(* IEC 61131-3 sources: SJ_AGV/PLC/Standard_functions.4.4.0/Navigation, 2 files *)

(* ---- LS2000_FB.ST ---- *)
FUNCTION_BLOCK LS2000_FB
VAR_EXTERNAL
	NDC8 : NDC8_T;
END_VAR

VAR_INPUT

END_VAR

VAR_OUTPUT
	Slowdown : bool;
END_VAR

VAR
	LS2000Field1TON :TON;
	LS2000Field2TON :TON;
END_VAR
(* Function to slow down, and eventually stop, if there is an obstacle in the path of the LS2000. *)

LS2000Field1TON (IN:= NDC8.LS2000.Field1_Triggered, PT:=T#160ms); (*Timer 160ms to filter signal*)
LS2000Field2TON (IN:= NDC8.LS2000.Field2_Triggered, PT:=T#160ms); (*Timer 160ms to filter signal *)

(* Stop window (Field 1), relative the scanner. *)
NDC8.LS2000.Field1_X1 := NDC8.LS2000.X - 100;	(* 500 mm behind. 		*)
NDC8.LS2000.Field1_X2 := NDC8.LS2000.X + 100;	(* 500 mm in front. 	*)
NDC8.LS2000.Field1_Y1 := NDC8.LS2000.Y - 100;	(* 500 mm to the left. 	*)
NDC8.LS2000.Field1_Y2 := NDC8.LS2000.Y + 100;	(* 500 mm to the right. *)

(* Slow down window (Field 2), relative the scanner. *)
NDC8.LS2000.Field2_X1 := NDC8.LS2000.X - 100;	(* 1000 mm behind.		*)
NDC8.LS2000.Field2_X2 := NDC8.LS2000.X + 100;	(* 1000 mm in front.	*)
NDC8.LS2000.Field2_Y1 := NDC8.LS2000.Y - 100;	(* 1000 mm to the left.	*)
NDC8.LS2000.Field2_Y2 := NDC8.LS2000.Y + 100;	(* 1000 mm to the right.*)

if INPUT.Manual  or NDC8.LoadOperation.OperationCode <> 0 then
	NDC8.LS2000.Field1_X1 := NDC8.LS2000.X ;	(* 500 mm behind. 		*)
	NDC8.LS2000.Field1_X2 := NDC8.LS2000.X;	(* 500 mm in front. 	*)
	NDC8.LS2000.Field1_Y1 := NDC8.LS2000.Y;	(* 500 mm to the left. 	*)
	NDC8.LS2000.Field1_Y2 := NDC8.LS2000.Y;	(* 500 mm to the right. *)

	NDC8.LS2000.Field2_X1 := NDC8.LS2000.X;	(* 1000 mm behind.		*)
	NDC8.LS2000.Field2_X2 := NDC8.LS2000.X;	(* 1000 mm in front.	*)
	NDC8.LS2000.Field2_Y1 := NDC8.LS2000.Y;	(* 1000 mm to the left.	*)
	NDC8.LS2000.Field2_Y2 := NDC8.LS2000.Y;	(* 1000 mm to the right.*)
end_if;

(* Stop the vehicle if it is about to run into a low hanging obstacle and hit the LS2000. *)
StopLS2000 := LS2000Field1TON.q or (NDC8.Position.NavLevel < 45 and INPUT.Auto = TRUE);
DisplayStopString(INStatus:=StopLS2000, StopString:=197, StopValue:=0);

(* Slow the vehicle down if it is about to run into a low hanging obstacle and hit the LS2000. *)
Slowdown := LS2000Field2TON.q  ;
DisplayStopString(INStatus:=Slowdown, StopString:=198, StopValue:=0);

END_FUNCTION_BLOCK

(* ---- NAVIGATION_FB.ST ---- *)
FUNCTION_BLOCK NAVIGATION_FB
VAR_EXTERNAL
	NDC8 : NDC8_T;
END_VAR

VAR_INPUT
	AutoInsertNotInsideTargetSafety : bool;
	ModePPA : bool;
END_VAR

VAR_OUTPUT

END_VAR

VAR
	NavMethod : NavMethod_FB;
	PreviousSegmentID,
	NavMethodState: DINT;
	SegmentChange,
	WheelSpinning,
	NavlevelTrigger : Bool;
	NavlevelTrigger_RT,
	PositionKnown_RT : F_trig;
	PositionKnown_FT : F_trig;

	WheelSpinningTimer,
	SegmentChangeTimer : TON;

END_VAR
(*
if ndc8.SegmentTrigger.Value > 0 then
	NDC8.VehicleNavigator.SetNavMethod := ndc8.SegmentTrigger.Value;
end_if;

Case NavMethodState of
0: if ndc8.SegmentTrigger.Value <> NDC8.VehicleNavigator.NavMethod then
		NavMethodState := 10;
	end_if;
10:	NavMethod();
	if NavMethod.Finished or NavMethod.ErrorCode > 0 or NDC8.SegmentTrigger.Value = 0 then
		NavMethodState := 0;
	end_if;
end_case;
*)

InStatus:=NavMethod.ErrorCode > 0;
DisplayStopString(INStatus:=InStatus, StopString:=53, StopValue:=0);							(* Undefined mode. *)

(* NAVIGATION init.				NOTE! Error codes > 5 is not supported in VMC500. *)

InStatus	:=	AutoInsertNotInsideTargetSafety
				and not NDC8.VehicleControl.Moving; ;
DisplayStopString(INStatus:=InStatus, StopString:=43, StopValue:=0);							(* Autoinsert *)

InStatus 	:= (NDC8.NavInit.Error = 1);
DisplayStopString(INStatus:=InStatus, StopString:=53, StopValue:=0);							(* Invalid init method *)

InStatus 	:= (NDC8.NavInit.Error = 3);
DisplayStopString(INStatus:=InStatus, StopString:=54, StopValue:=0);							(* Target don't exist *)

InStatus 	:= (NDC8.NavInit.Error = 4);
DisplayStopString(INStatus:=InStatus, StopString:=166, StopValue:=0);							(* Not supported *)

InStatus 	:= (NDC8.NavInit.Error = 5);
DisplayStopString(INStatus:=InStatus, StopString:=66, StopValue:=0);							(* not in manual mode or semi manual *)

InStatus 	:= (NDC8.NavInit.Error = 6);
DisplayStopString(INStatus:=InStatus, StopString:=168, StopValue:=0);							(* too few reflector bearings *)

InStatus 	:= (NDC8.NavInit.Error = 7);
DisplayStopString(INStatus:=InStatus, StopString:=144, StopValue:=0);							(* bad distribution of bearings *)

InStatus 	:= (NDC8.NavInit.Error = 8);
DisplayStopString(INStatus:=InStatus, StopString:=145, StopValue:=0);							(* reflector init failed in current search area *)

InStatus 	:= (NDC8.NavInit.Error = 9);
DisplayStopString(INStatus:=InStatus, StopString:=169, StopValue:=0);							(* ambiguous position (more than one valid position in current search area) *)

InStatus 	:= (NDC8.NavInit.Error = 10);
DisplayStopString(INStatus:=InStatus, StopString:=170, StopValue:=0);							(* init calculation aborted *)

InStatus 	:= (NDC8.NavInit.Error = 11);
DisplayStopString(INStatus:=InStatus, StopString:=171, StopValue:=0);							(* agv is moving *)

InStatus 	:= (NDC8.NavInit.Error = 12);
DisplayStopString(INStatus:=InStatus, StopString:=172, StopValue:=0);							(* position outside search area *)

InStatus 	:= (NDC8.NavInit.Error = 15);
DisplayStopString(INStatus:=InStatus, StopString:=173, StopValue:=0);							(* no range measurements *)

InStatus 	:= (NDC8.NavInit.Error = 16);
DisplayStopString(INStatus:=InStatus, StopString:=174, StopValue:=0);							(* bad range match *)

InStatus 	:= (NDC8.NavInit.Error = 17);
DisplayStopString(INStatus:=InStatus, StopString:=191, StopValue:=0);							(* empty init area *)

InStatus 	:= (NDC8.NavInit.Error = 18);
DisplayStopString(INStatus:=InStatus, StopString:=192, StopValue:=0);							(* multi oriented point *)

(* DETECT A VEHICLE WHICH IS STUCK
With the NDC8 2.7 release introduced new parameters, which can be used for detecting a spinning wheel from the PLC. *)

WheelSpinning := ABS(NDC8.VehicleNavigator.CorrectionX) > 100;			(* If correcting above this value, for more than 10 seconds, *)
WheelSpinningTimer(IN:=WheelSpinning, PT:= t#10s);

SegmentChange := PreviousSegmentID <> NDC8.LayoutPosition.Segment;		(* ...or does not change segment ID after two minutes *)
SegmentChangeTimer(IN:=SegmentChange, PT:= t#120s);
PreviousSegmentID := NDC8.LayoutPosition.Segment;

if NDC8.LayoutPosition.InSystem											(* ...when driving in automatic mode. *)
	and NDC8.Automatic.ExecDriveCommand
	and NDC8.VehicleControl.OperationMode = 0
	and NDC8.VehicleControl.SetSpeed <> 0
	and NDC8.VehicleControl.Moving
	and (WheelSpinningTimer.q or SegmentChangeTimer.q) then
      			StopSpinningWheel := true;								(* ...then stop the vehicle to avoid burning the motor and the wheel! *)
elsif Input.Reset_PB then                    (* Reset of the stop *)
    StopSpinningWheel := false;
end_if;

(* Display update *)
DisplayStopString(INStatus:=StopSpinningWheel, StopString:=86, StopValue:=0);

END_FUNCTION_BLOCK
